PROGRAM TelescopeControl
VAR_INPUT
(*
TCS interface section
see https://gitlab.aip.de/bmk10k/telescope_firmware/snippets/5
*)
	
	// boolean, true: Power on, false: power off
	power: 		BOOL;
	// boolean, true: go to home position, unset track/goto if active
	gohome: 	BOOL;
	// boolean, true: go into park position, ready to stow telescope, unset track/goto
	park: 		BOOL;
	// boolean, TRUE: MOVE telescope TO last ra/de AND start tracking. Set 'goto' TO FALSE, IF TRUE. FALSE: Stop tracking as soon as possible
	track: 		BOOL;
	// boolean, TRUE: MOVE telescope TO tau/de AND stop there. Set track TO FALSE, IF TRUE. FALSE: no effect.)
	goto:		BOOL;	
	// move the telescope to a given az-alt position
	slew:		BOOL;
	// boolean, TRUE: Stop motion OF telescope immediately, set goto AND track TO FALSE. FALSE: Allow motion OF telescope again via track/goto).
	stop:		BOOL;	
	// initiates reset on all axis
	reset:		BOOL;
	// automatic tracking after goto
	autotrack:	BOOL := TRUE;
	// apparent right ascension, degrees, double
	rightascension:		LREAL := (4.0 + 35.0/60.0 + 54.09/3600.0) *15.0;	
	// apparent declination, degrees, double
	declination: 		LREAL := 16.0 + 30.0/60.0 + 25.4/3600.0;
	// desired elevation of the telescope pointing 
	elevation:	LREAL := 45.0;
	// desired azimut of the telescope pointing 
	azimuth:	LREAL := 320.0;
	// absolute offset for elevation
	elevation_offset:	LREAL := 0.0;
	// absolute offset for azimuth
	azimuth_offset : 	LREAL := 0.0;
	// absolute offset for time
	time_offset: 		LREAL := 0.0;
	// Nasmyth port 1 or 2
	Nasmyth_port: 		USINT;
END_VAR
VAR
	// actual command from the TCS
	TCS_command: 	E_TCSCommand;
	// current Julian Date calculated from system time
	jd:				LREAL;
	// local siderial time calculated from Julian date
	lst:			LREAL;
	// elevation calulated when ra and dec are set by TCS
	elevation_calc:	LREAL; 
	// azimuth calulated when ra and dec are set by TCS
	azimuth_calc:	LREAL;
	// right ascension calulated when azimuth and elevation are set by TCS
	rightascension_calc:	LREAL;
	// declination calulated when azimuth and elevation are set by TCS
	declination_calc:		LREAL;
	// hour angle
	Hourangle_calc: LREAL;
	// precise astronomical	time
	fbTime: FB_AstroClock;
	
	eq2hor2:	FB_EQ2HOR2;
	hor2eq:		FB_HOR2EQ;
	
	// triggers power-failure event
	powerfailure: 	BOOL;
	// triggers power warning
	poweronwarning:	TP;
	// power on timeout
	power_timeout:	TON;
	// tracking delay
	tracking_delay:	TON;
	// telescope is parked
	isparked:		BOOL;
	TCSpowerEvent,
	TCSgohomeEvent,
	TCSparkEvent,
	TCSgotoEvent,
	TCStrackEvent,
	TCSstopEvent,
	AltitudeEvent,
	TCSreadyEvent: FB_Eventlog;
	MQTTTimer : TON := (PT:=T#5S);
	// rotational velocity of the elevation
	ElevationVelocity: LREAL;
	// rotational velocity of the elevation
	AzimuthVelocity: LREAL;
	// sign of derotation
	StatusWord, LastStatus:	UDINT;
	ignore_covers:	BOOL;
END_VAR
VAR_OUTPUT
	//		TRUE, IF telescope can be operated
	ready:		BOOL; 
	// indicates an error on one of the components
	error:		BOOL;	
	//error id of axis
	errorid:	UDINT;	
	//TRUE, IF telescope is in fast-MOVE phase (includes pole-swap)
	sliding:	BOOL;	
	//TRUE, IF telescope is on tracking position AND currently tracking.
	tracking:	BOOL;	
	//TRUE, IF telescope is AT rest.
	stopped:	BOOL;	
	// true position of the elevation
	elevation_current:	LREAL;
	// true position of the azimuth
	azimuth_current:	LREAL;
	//	(time in sec. to reach the goto/track position)
	slewtime:			LREAL; 
	// True: telescope is calibrated
	homed:				BOOL;
	// telescope does not accept further commands
	busy:				BOOL;
END_VAR
VAR CONSTANT
// STELLA1
	// telescope site longitude, source: Google 
	longitude: 		LREAL := -16.50926; //13.101867;
	// telescope site latitude, source: Google
	latitude: 		LREAL := 28.30120; //52.404940;
	// telescope site height above sea level: estimated
	altitude: 		LREAL := 2390.0;
	elevation_park: LREAL := 60.0;
	azimuth_park: 	LREAL := 0.0;
	
	elevation_home: LREAL := 55.0;
	azimuth_home: 	LREAL := 180.0;
END_VAR
VAR PERSISTENT
	// azimuth axis offset/misalignment north-south
	AN_E:	LREAL;
	// azimuth axis offset/misalignment east-west
	AE_E:	LREAL;
	// gravitational flexure correction at the horizon
	TF:		LREAL;
	// collimation error of the electromagnetic axis
	BNP:	LREAL;
	// azimuth axis offset/misalignment north-south
	AN_A:	LREAL;
	// azimuth axis offset/misalignment east-west,
	AE_A:	LREAL;
	// Non-perpendicularity between the mount azimuth and elevation axes
	NPAE:	LREAL;
END_VAR

TelescopeAuxiliary();

// get the system time
fbTime();
jd := DateTime2JD(fbTime.time_RTCEX2);
lst := CT2LST(longitude, jd);
// set reset state either by hardware (key pressed) or by software (set by e.g. tcs)
IF GVL_Main.reset_switch THEN
	reset := TRUE;
END_IF


IF ElevationControl.error THEN
	errorid := ElevationControl.ErrorID;
	ElevationControl.reset := reset;
ELSIF AzimuthElevationControl.error THEN
	errorid := AzimuthElevationControl.ErrorID;
	AzimuthElevationControl.Reset := reset;
END_IF

error := ElevationControl.error OR 
		 AzimuthElevationControl.error;

slewtime := MAX(ElevationControl.slewtime, AzimuthElevationControl.slewtime);
			
IF error THEN
	gohome := 	FALSE;
	track := 	FALSE;
	goto := 	FALSE;
	slew := 	FALSE;
ELSE
	errorid := 0;
END_IF

IF ElevationControl.error THEN
	ElevationControl.enable := FALSE;
	AzimuthElevationControl.enable := FALSE;
	HydraulicsControl.close_brake();
END_IF

eq2hor2(alpha := rightascension,
	delta := declination,
	lon := longitude,
	lat := latitude,
	JD := jd + time_offset,
	alt => elevation_calc,
	az => azimuth_calc,
	ha => hourangle_calc);

// apply pointing model
elevation_calc := elevation_calc + PointingModelElevation(azimuth_calc, elevation_calc, elevation_offset, AN_E, AE_E, TF);
azimuth_calc := azimuth_calc + PointingModelAzimuth(azimuth_calc, elevation_calc, azimuth_offset, BNP, AN_A, AE_A, NPAE);
ElevationVelocity := F_Elevationvelocity(azimuth_calc, latitude);
AzimuthVelocity := F_Azimuthvelocity(elevation_calc, azimuth_calc, latitude);

IF (azimuth_calc > 350.0 AND AzimuthVelocity > 0.0) OR (azimuth_calc > 440.0) THEN
	azimuth_calc := azimuth_calc - 360.0;
ELSIF (azimuth_calc < -10.0 AND AzimuthVelocity < 0.0) OR (azimuth_calc < -50.0) THEN
	azimuth_calc := azimuth_calc + 360.0;
END_IF

// get current coordinates	
azimuth_current := AzimuthElevationControl.act_position;
elevation_current := ElevationControl.actual_position;

// calculate equatorial coordinates
hor2eq(alt := elevation_current - PointingModelElevation(azimuth_calc, elevation_calc, elevation_offset, AN_E, AE_E, TF), 
		az := azimuth_current - PointingModelAzimuth(azimuth_calc, elevation_calc, azimuth_offset, BNP, AN_A, AE_A, NPAE),
		jd := jd,
		lat := latitude,
		lon := longitude,
		altitude := altitude,
		ra => rightascension_calc,
		dec => declination_calc);		
	
poweronwarning(IN := power, PT := T#10S);

power_timeout(IN := TCS_command = E_TCSCommand.no_command AND NOT isparked, PT := T#12H);
IF power_timeout.Q AND NOT isparked AND ready THEN
	park := TRUE;
END_IF

// set TCS_command according to state variables ordered by precedence
IF power THEN
	TCS_command := E_TCSCommand.poweron;
ELSIF stop THEN
	TCS_command := E_TCSCommand.stop;
	goto := FALSE;
	track := FALSE;
	slew := FALSE;
	gohome := FALSE;
	park := FALSE;
ELSIF park THEN
	goto := FALSE;
	track := FALSE;
	slew := FALSE;
	IF ready AND stopped THEN
		TCS_command := E_TCSCommand.park;
	END_IF
ELSIF gohome THEN
	goto := FALSE;
	track := FALSE;
	slew := FALSE;
	IF ready AND NOT busy AND stopped THEN
		TCS_command := E_TCSCommand.gohome;
	END_IF
ELSIF goto THEN
	track := FALSE;
	slew := FALSE;
	IF ready AND NOT busy THEN
		TCS_command := E_TCSCommand.goto;
	END_IF
ELSIF slew THEN
	goto := FALSE;
	track := FALSE;
	IF ready AND NOT busy THEN
		TCS_command := E_TCSCommand.slew;
	END_IF
ELSIF track THEN
	goto := FALSE;
	slew := FALSE;
	IF ready AND NOT busy THEN
		TCS_command := E_TCSCommand.track;
	END_IF
ELSE
	TCS_command := E_TCSCommand.no_command;
	ElevationControl.MoveAxis := FALSE;
	AzimuthElevationControl.MoveAxis := FALSE;
	ElevationControl.Tracking := FALSE;
	AzimuthElevationControl.Tracking := FALSE;
END_IF

IF TCS_command = E_TCSCommand.poweron THEN
	poweron();
ELSIF TCS_command = E_TCSCommand.stop THEN
	stoptelescope();
ELSIF TCS_command = E_TCSCommand.park THEN
	parktelescope();
ELSIF TCS_command = E_TCSCommand.gohome THEN
	hometelescope();
ELSIF TCS_command = E_TCSCommand.goto THEN
	gototelescope();
ELSIF TCS_command = E_TCSCommand.slew THEN
	slewtelescope();
ELSIF TCS_command = E_TCSCommand.track THEN
	tracktelescope();
END_IF
 
sliding := NOT tracking AND (ElevationControl.ElevationAxis.InMotion OR ElevationControl.ElevationAxis.InRamp OR
			AzimuthElevationControl.AzimuthAxis.InMotion OR AzimuthElevationControl.AzimuthAxis.InRamp);

// signal must be stable for 3000MS			
tracking_delay(in := ElevationControl.ElevationAxis.isTracking AND 
			AzimuthElevationControl.AzimuthAxis.isTracking,PT :=T#5500MS, Q => tracking);
			
stopped :=  (NOT ElevationControl.enable OR ElevationControl.ElevationAxis.StandStill) AND 
			(NOT AzimuthElevationControl.Enable OR AzimuthElevationControl.AzimuthAxis.StandStill);
			
homed := ElevationControl.Calibrated AND
			AzimuthElevationControl.calibrated;
			
ready := homed AND 
	(CoverControl.isopen OR ignore_covers) AND 
	ElevationControl.enable AND
	AzimuthElevationControl.enable AND HydraulicsControl.brake_open AND 
    NOT error;

busy := ElevationControl.ElevationAxis.Busy OR
		AzimuthElevationControl.AzimuthAxis.Busy;
// unset the STOP command if telescope is already stopped
IF stopped THEN
	stop := FALSE;
END_IF
	
IF NOT error THEN
	reset := FALSE;
END_IF

IF SafetyHandling.Emergency_stop THEN
	ElevationControl.enable := FALSE;
	AzimuthElevationControl.enable := FALSE;
END_IF
IF sliding OR track OR tracking THEN
	MQTTTimer.PT := T#1000MS;
ELSE
	MQTTTimer.PT := T#5000MS;
END_IF
MQTTTimer(IN:=TRUE);
IF MQTTTimer.Q THEN // publish new payload every second
	MQTTTimer(IN:=FALSE);

	MAIN.MQTTClient.Publish('telescope', 'dome', 'JulianDate', LREAL_TO_STRING(jd));
	MAIN.MQTTClient.Publish('telescope', 'dome', 'LocalSiderialTime', LREAL_TO_STRING(lst));
	MAIN.MQTTClient.Publish('telescope', 'dome', 'Azimuth', LREAL_TO_STRING(azimuth_current));
	MAIN.MQTTClient.Publish('telescope', 'dome', 'Elevation', LREAL_TO_STRING(elevation_current));
	MAIN.MQTTClient.Publish('telescope', 'dome', 'HourAngle', LREAL_TO_STRING(hourangle_calc));
	MAIN.MQTTClient.Publish('telescope', 'dome', 'RightAscension', LREAL_TO_STRING(rightascension_calc));
	MAIN.MQTTClient.Publish('telescope', 'dome', 'Declination', LREAL_TO_STRING(declination_calc));
	MAIN.MQTTClient.Publish('telescope', 'dome', 'azimuth_offset', LREAL_TO_STRING(azimuth_offset));
	MAIN.MQTTClient.Publish('telescope', 'dome', 'elevation_offset', LREAL_TO_STRING(elevation_offset));
	MAIN.MQTTClient.Publish('telescope', 'dome', 'elevation_torque', LREAL_TO_STRING(ElevationControl.elevation_torque));
	MAIN.MQTTClient.Publish('telescope', 'dome', 'azimuth_torque', LREAL_TO_STRING(AzimuthElevationControl.azimuth_torque));
	
	MAIN.MQTTClient.Publish('telescope', 'dome', 'errorid',		UDINT_TO_STRING(errorid));
	MAIN.MQTTClient.Publish('telescope', 'dome', 'error',		BOOL_TO_STRING(error));
	MAIN.MQTTClient.Publish('telescope', 'dome', 'ready',		BOOL_TO_STRING(ready));
	MAIN.MQTTClient.Publish('telescope', 'dome', 'busy',		BOOL_TO_STRING(busy));
	MAIN.MQTTClient.Publish('telescope', 'dome', 'sliding',		BOOL_TO_STRING(sliding));
	MAIN.MQTTClient.Publish('telescope', 'dome', 'tracking', 	BOOL_TO_STRING(tracking));
	MAIN.MQTTClient.Publish('telescope', 'dome', 'stopped',		BOOL_TO_STRING(stopped));
	MAIN.MQTTClient.Publish('telescope', 'dome', 'homed',		BOOL_TO_STRING(homed));
END_IF

StatusWord.0 := error;
StatusWord.1 := ready;
StatusWord.2 := sliding;
StatusWord.3 := tracking;
StatusWord.4 := stopped;
StatusWord.5 := homed;
StatusWord.6 := power;
StatusWord.7 := park;
StatusWord.8 := gohome;
StatusWord.9 := track;
StatusWord.10 := goto;
StatusWord.11 := slew;
StatusWord.12 := stop;
StatusWord.13 := busy;

IF StatusWord<>LastStatus THEN // publish new payload every second
	LastStatus := StatusWord;
	MAIN.MQTTClient.Publish('telescope', 'dome', 'error',		BOOL_TO_STRING(error));
	MAIN.MQTTClient.Publish('telescope', 'dome', 'ready',		BOOL_TO_STRING(ready));
	MAIN.MQTTClient.Publish('telescope', 'dome', 'sliding',		BOOL_TO_STRING(sliding));
	MAIN.MQTTClient.Publish('telescope', 'dome', 'tracking', 	BOOL_TO_STRING(tracking));
	MAIN.MQTTClient.Publish('telescope', 'dome', 'stopped',		BOOL_TO_STRING(stopped));
	MAIN.MQTTClient.Publish('telescope', 'dome', 'homed',		BOOL_TO_STRING(homed));
	MAIN.MQTTClient.Publish('telescope', 'dome', 'power',		BOOL_TO_STRING(power));
	MAIN.MQTTClient.Publish('telescope', 'dome', 'park',		BOOL_TO_STRING(park));
	MAIN.MQTTClient.Publish('telescope', 'dome', 'gohome',		BOOL_TO_STRING(gohome));
	MAIN.MQTTClient.Publish('telescope', 'dome', 'track',		BOOL_TO_STRING(track));
	MAIN.MQTTClient.Publish('telescope', 'dome', 'goto',		BOOL_TO_STRING(goto));
	MAIN.MQTTClient.Publish('telescope', 'dome', 'slew',		BOOL_TO_STRING(slew));
	MAIN.MQTTClient.Publish('telescope', 'dome', 'stop',		BOOL_TO_STRING(stop));
	MAIN.MQTTClient.Publish('telescope', 'dome', 'busy',		BOOL_TO_STRING(busy));
END_IF


(* Event function blocks start here. *)
TCSpowerEvent(	Trigger := powerfailure, 
				Level := ADSLOG_MSGTYPE_ERROR,
				FormatString := 'power %s',
				OnMessage := 'Failure',
				OffMessage := 'OK');

TCSgohomeEvent(	Trigger := gohome, 
				Level := ADSLOG_MSGTYPE_HINT,
				FormatString := 'GOHOME %s',
				OnMessage := 'commencing',
				OffMEssage := 'completed');
TCSparkEvent(	Trigger := park, 
				Level := ADSLOG_MSGTYPE_HINT,
				FormatString := 'PARK %s',
				OnMessage := 'commencing',
				OffMEssage := 'completed');
TCSgotoEvent(	Trigger := goto, 
				Level := ADSLOG_MSGTYPE_HINT,
				FormatString := 'GOTO %s',
				OnMessage := 'commencing',
				OffMEssage := 'completed');
TCStrackEvent(	Trigger := track, 
				Level := ADSLOG_MSGTYPE_HINT,
				FormatString := 'TRACK %s',
				OnMessage := 'commencing',
				OffMEssage := 'completed');
TCSstopEvent(	Trigger := stop, 
				Level := ADSLOG_MSGTYPE_WARN,
				FormatString := 'STOP %s',
				OnMessage := 'commencing',
				OffMEssage := 'completed',
				OffLevel := ADSLOG_MSGTYPE_HINT);
AltitudeEvent(	Trigger := power AND elevation_calc<0.0, 
				Level := ADSLOG_MSGTYPE_WARN,
				FormatString := '%s',
				OnMessage := 'Target below horizon',
				OffMEssage := '');
TCSreadyEvent(	Trigger := power AND ready, 
				Level := ADSLOG_MSGTYPE_HINT,
				FormatString := '%s',
				OnMessage := 'STELLA1 startup finished');

METHOD gototelescope: USINT
VAR_INPUT
END_VAR
VAR
	GoToEvent:	FB_Eventlog;
	command_timeout:	TON;
END_VAR
VAR_STAT
	Stage:		USINT := 0;
	LastStage:	USINT := 101;
END_VAR
gototelescope := Stage;
command_timeout(IN := Stage < 100, PT := T#600S);
IF command_timeout.Q THEN
	error := TRUE;
	errorid := 16#10;
	goto := FALSE;
	Stage := 0;
	RETURN;
END_IF

IF elevation_calc<2.0 THEN
	error := TRUE;
	errorid := 16#15;
	goto := FALSE;
	Stage := 0;
	RETURN;
END_IF

IF reset OR error THEN
	Stage := 0;
	RETURN;
END_IF

CASE Stage OF
	0:	
		IF ready AND NOT busy THEN
			Stage := 25;
		END_IF
	25:	
		ElevationControl.position := elevation_calc;
		AzimuthElevationControl.position := azimuth_calc;
		ElevationControl.velocity := 5.0;
		AzimuthElevationControl.velocity := 10.0;
		
		ElevationControl.MoveAxis := TRUE;
		AzimuthElevationControl.MoveAxis := TRUE;
		IF ElevationControl.ElevationAxis.Busy AND
			AzimuthElevationControl.AzimuthAxis.Busy THEN
				Stage := 50;
		END_IF
	50:
		IF NOT ElevationControl.ElevationAxis.Busy AND ElevationControl.ElevationAxis.MoveDone THEN
			ElevationControl.MoveAxis := FALSE;
		END_IF
		IF NOT AzimuthElevationControl.AzimuthAxis.Busy AND AzimuthElevationControl.AzimuthAxis.MoveDone THEN
			AzimuthElevationControl.MoveAxis := FALSE;
		END_IF
		IF NOT ElevationControl.MoveAxis AND 
           NOT AzimuthElevationControl.MoveAxis THEN
		   Stage := 75;
		END_IF
	75:
		IF NOT sliding AND stopped THEN // all axis standstill
			Stage := 100;
		END_IF
	100:
		ElevationControl.MoveAxis := FALSE;
		AzimuthElevationControl.MoveAxis := FALSE;
		azimuth := azimuth_calc;
		elevation := elevation_calc;
		goto := FALSE;
		// enable automatic tracking
		track := autotrack;
		Stage := 0;
END_CASE
GoToEvent(Trigger := Stage > LastStage, FormatString := 'GoTo progress: %s', OnMessage := USINT_TO_STRING(Stage));
LastStage := Stage;
END_METHOD

METHOD hometelescope : BOOL
VAR_INPUT
END_VAR

VAR
	HomeEvent: FB_Eventlog;
	command_timeout: TON;
END_VAR
command_timeout(IN := NOT hometelescope, PT := T#600S);
IF command_timeout.Q THEN
	error := TRUE;
	errorid := 16#30;
	hometelescope :=TRUE;
END_IF

IF ready AND stopped AND NOT busy AND NOT tracking THEN
	ElevationControl.velocity := 5.0;
	ElevationControl.position := elevation_home;
	ElevationControl.MoveAxis := TRUE;
	AzimuthElevationControl.velocity := 10.0;
	AzimuthElevationControl.position := azimuth_home;
	AzimuthElevationControl.MoveAxis := TRUE;
END_IF

IF ElevationControl.ElevationAxis.MoveDone AND 
	AzimuthElevationControl.AzimuthAxis.MoveDone THEN 
	gohome := FALSE;
	elevation := elevation_current;
	azimuth := azimuth_current;
	hometelescope := TRUE;
ELSE
	hometelescope := FALSE;
END_IF

HomeEvent(Trigger := hometelescope, 
			Level := ADSLOG_MSGTYPE_HINT,
			FormatString := '%s',
			OnMessage := 'Telescope is homed.');
END_METHOD

METHOD parktelescope: USINT
VAR_INPUT
END_VAR
VAR
	ParkEvent:	FB_Eventlog;
	command_timeout:	TON;
END_VAR
VAR_STAT
	Stage:		USINT := 0;
	LastStage:	USINT := 101;
END_VAR
parktelescope := Stage;
command_timeout(IN := Stage < 100, PT := T#600S);
IF command_timeout.Q THEN
	error := TRUE;
	errorid := 16#20;
	Stage := 0;
END_IF
IF reset OR error THEN
	Stage := 0;
END_IF
IF isparked THEN
	Stage := 100;
END_IF
CASE Stage OF
	0: 
		gohome := 	FALSE;
		track := 	FALSE;
		goto := 	FALSE;
		slew := 	FALSE;
		IF Error THEN // emergency park
			HydraulicsControl.close_brake();
			ElevationControl.enable := FALSE;
			AzimuthElevationControl.Enable := FALSE;
			CoverControl.close := TRUE;	
			Stage := 80;
		END_IF
		Stage := 20;
	20:
		ElevationControl.position := elevation_park;
		ElevationControl.velocity := 10.0;
		ElevationControl.MoveAxis := TRUE;
		AzimuthElevationControl.position := azimuth_park;
		AzimuthElevationControl.velocity := 10;
		AzimuthElevationControl.MoveAxis := TRUE;
		IF ElevationControl.ElevationAxis.Busy AND
			AzimuthElevationControl.AzimuthAxis.Busy THEN
				Stage := 40;
		END_IF
	40:
		IF ElevationControl.ElevationAxis.MoveDone THEN
			ElevationControl.MoveAxis := FALSE;
		END_IF
		IF AzimuthElevationControl.AzimuthAxis.MoveDone THEN
			AzimuthElevationControl.MoveAxis := FALSE;
		END_IF
		IF NOT sliding THEN // all axis standstill
			Stage := 60;
		END_IF
	60:
		IF stopped THEN 
			ElevationControl.enable := FALSE;
			AzimuthElevationControl.Enable := FALSE;
			Stage := 80;
		END_IF
		
		ElevationControl.MoveAxis := FALSE;
		AzimuthElevationControl.MoveAxis := FALSE;
	80:
		IF HydraulicsControl.brake_closed THEN
			CoverControl.close := TRUE;			
		END_IF
		IF CoverControl.isclosed THEN
			Stage := 100;
		END_IF
	100:
			isparked := TRUE;
			park := FALSE;
			parktelescope := 100;
			Stage := 0;	
END_CASE
ParkEvent(Trigger := Stage > LastStage, FormatString := 'Parking progress: %s', OnMessage := USINT_TO_STRING(Stage));
LastStage := Stage;
END_METHOD

METHOD poweron : BOOL
VAR_INPUT
END_VAR
VAR
END_VAR
IF NOT Main.brake_clearing THEN
	powerfailure := TRUE;
	TCSpowerEvent.OnMessage := 'failure: brake clearing not set';
	power := FALSE;
ELSIF NOT Transformer.power_OK THEN
	powerfailure := TRUE;
	TCSpowerEvent.OnMessage := 'failure: main power failure';
	power := FALSE;
ELSIF NOT Transformer.phase_available THEN
	powerfailure := TRUE;
	TCSpowerEvent.OnMessage := 'failure: hydraulics power failure';
	power := FALSE;
ELSIF error THEN
	powerfailure := TRUE;
	TCSpowerEvent.OnMessage := 'Generic error during power on occured.';
	power := FALSE;
ELSE
	powerfailure := FALSE;		
END_IF
// COVER MUST BE OPENED FOR A SUCCESSFUL WAKE & SHAKE COMMAND!
Covercontrol.open := TRUE;

// enable elevation, enable azimuth
IF MAIN.ready AND CoverControl.isopen THEN
	ElevationControl.enable := TRUE;
	AzimuthElevationControl.enable := TRUE;
END_IF

IF ElevationControl.Ready AND NOT ElevationControl.Calibrated THEN
	ElevationControl.HomeAxis := TRUE;
END_IF

IF AzimuthElevationControl.ready AND NOT AzimuthElevationControl.calibrated THEN
	AzimuthElevationControl.HomeAxis := TRUE;
END_IF

// start calibration of focus after elevation has been calibrated
// this avoids imbalance by the M2 mirror on the elvation during its calibration

IF CoverControl.isopen AND 
	ElevationControl.Calibrated AND ElevationControl.Ready AND
	AzimuthElevationControl.calibrated AND AzimuthElevationControl.ready THEN
	power := FALSE;
	poweron := TRUE;
	isparked := FALSE;
	// slew the telescope to the home position
	gohome := TRUE;
ELSE
	poweron := FALSE;
END_IF
END_METHOD

METHOD slewtelescope : USINT
VAR_INPUT
END_VAR
VAR
	SlewEvent:	FB_Eventlog;
	command_timeout: TON;
END_VAR
VAR_STAT
	Stage:		USINT := 0;
	LastStage:	USINT := 101;
END_VAR
slewtelescope := Stage;
command_timeout(IN := Stage < 100, PT := T#600S);
IF command_timeout.Q THEN
	error := TRUE;
	errorid := 16#40;
	slew := FALSE;
	Stage := 0;
END_IF
IF reset OR error THEN
	Stage := 0;
END_IF
CASE Stage OF
	0:	
		IF ready AND stopped AND NOT busy AND NOT tracking THEN
			Stage := 25;
		END_IF
	25:
		ElevationControl.position := elevation;
		ElevationControl.velocity := 5.0;
		ElevationControl.MoveAxis := TRUE;
		AzimuthElevationControl.position := azimuth;
		AzimuthElevationControl.velocity := 10.0;
		AzimuthElevationControl.MoveAxis := TRUE;
		IF ElevationControl.ElevationAxis.Busy AND
			AzimuthElevationControl.AzimuthAxis.Busy THEN
				Stage := 50;
		END_IF
	50:
		IF ElevationControl.ElevationAxis.MoveDone THEN
			ElevationControl.MoveAxis := FALSE;
		END_IF
		
		IF AzimuthElevationControl.AzimuthAxis.MoveDone THEN
			AzimuthElevationControl.MoveAxis := FALSE;
		END_IF

		IF NOT sliding AND stopped THEN // all axis standstill
			Stage := 100;
		END_IF
	100:
		ElevationControl.MoveAxis := FALSE;
		AzimuthElevationControl.MoveAxis := FALSE;
		rightascension := rightascension_calc;
		declination := declination_calc;
		slew := FALSE;
		Stage := 0;
END_CASE
SlewEvent(Trigger := Stage > LastStage, FormatString := 'Slew progress: %s', OnMessage := USINT_TO_STRING(Stage));
LastStage := Stage;
END_METHOD

METHOD stoptelescope : BOOL
VAR_INPUT
END_VAR
ElevationControl.StopAxis := TRUE;
AzimuthElevationControl.StopAxis := TRUE;
IF stopped THEN
	ElevationControl.StopAxis := FALSE;
	AzimuthElevationControl.StopAxis := FALSE;
	stop := FALSE;
END_IF
END_METHOD

METHOD tracktelescope : BOOL
VAR_INPUT
END_VAR
// Elevation
ElevationVelocity := F_Elevationvelocity(azimuth_calc, latitude);
AzimuthVelocity := F_Azimuthvelocity(elevation_calc, azimuth_calc, latitude);
IF elevation_current < 5.0 OR elevation_current > 89.5 THEN 
	track := FALSE;
END_IF
IF azimuth_current > 440.0 THEN
	track := FALSE;
END_IF

ElevationControl.position := elevation_calc;
IF NOT ElevationControl.Tracking THEN
	ElevationControl.velocity := 10.0;
	ElevationControl.MoveAxis := TRUE;
	IF NOT ElevationControl.ElevationAxis.Busy AND ElevationControl.ElevationAxis.MoveDone THEN
		ElevationControl.MoveAxis := FALSE;
		IF ElevationControl.ElevationAxis.isTracking THEN
			ElevationControl.velocity := ElevationVelocity;
		ELSE
			ElevationControl.velocity := 3.0*ElevationVelocity;
		END_IF
		ElevationControl.velocity := ElevationVelocity;
		ElevationControl.Tracking := TRUE;
	END_IF
ELSE
	ElevationControl.velocity := ElevationVelocity;
END_IF

// Azimuth
AzimuthElevationControl.position := azimuth_calc;
IF NOT AzimuthElevationControl.Tracking THEN
	AzimuthElevationControl.velocity := 10.0;
	AzimuthElevationControl.MoveAxis := TRUE;
	IF NOT AzimuthElevationControl.AzimuthAxis.Busy AND AzimuthElevationControl.AzimuthAxis.MoveDone THEN
		AzimuthElevationControl.MoveAxis := FALSE;
		IF AzimuthElevationControl.AzimuthAxis.isTracking THEN
			AzimuthElevationControl.velocity := AzimuthVelocity;
		ELSE
			AzimuthElevationControl.velocity := 3.0*AzimuthVelocity;
		END_IF
		AzimuthElevationControl.velocity := AzimuthVelocity;
		AzimuthElevationControl.Tracking := TRUE;
	END_IF
ELSE
	AzimuthElevationControl.velocity := AzimuthVelocity;
END_IF
END_METHOD

END_PROGRAM

(* stored: Version 1.1.0.1, ProductVersion 3.1.4024.9
   POU TelescopeControl: Id {6a4f2e3a-c9ee-4352-b4f6-4f9d94b2c472}, SpecialFunc None
   Method gototelescope: Id {c7053474-39ba-4cc3-ab24-2521b02cf8f4}
   Method hometelescope: Id {2c96c3e4-ffc4-4f92-b3af-46d302446b40}
   Method parktelescope: Id {99ae1f40-9696-469a-b290-774914abbb25}
   Method poweron: Id {34114692-caf6-4cf5-8270-8b1671f5dd0a}
   Method slewtelescope: Id {e66a400f-15f7-407b-9ae1-f4d90da8099d}
   Method stoptelescope: Id {3ed2c63a-7819-48f1-a5e6-de7431397407}
   Method tracktelescope: Id {8d4fcfbf-479d-4826-a883-1021b018a460} *)
